FUNCTION_BLOCK COLOR_SAT (* Compute Color Saturation *)
  (* Standard: 61499-1 *)
  (* Version 0.1, 2001-06-03, JHC, Rockwell Automation, XML version *)
  (* Version 0.0, 2000-01-10, JHC, Rockwell Automation, SRC version *)
  (* Compiler header: package fb.rt.hmi; *)
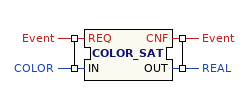
  EVENT_INPUT
    REQ WITH IN; (* Normal Execution Request *)
  END_EVENT
  EVENT_OUTPUT
    CNF WITH OUT; (* Execution Confirmation *)
  END_EVENT
  VAR_INPUT
    IN : COLOR;
  END_VAR
  VAR_OUTPUT
    OUT : REAL; (* Color saturation value *)
  END_VAR
  ALGORITHM REQ IN JAVA:
private float[]hsbvals=new float[3];
protected void service_REQ(boolean ei){
java.awt.Color c=IN.value;
hsbvals=java.awt.Color.RGBtoHSB(c.getRed(),c.getGreen(),c.getBlue(),hsbvals);
OUT.value=hsbvals[1];
CNF.serviceEvent(this);
}
  END_ALGORITHM
END_FUNCTION_BLOCK
